Staubli VAL3: FNearJt.pgx

public program FNearJt(joint j_Position, num n_Tolerance, bool& m_inRange[])
begin
  //判断当前位置是否在某关节点附近
  m_inRange=(abs(herej()-j_Position)<{1,1,1,2,2,2})

end
